TYPE (* IEC61131-3, Table 14#5 *)
  (* Standard: 1131-3 *)
  (* Version 0.0, 1/8/2024, Cheyan, Schneider Electric, Template *)
  PACKAGE Main;
  {SET_ATTRIBUTE(nxtDataType, /vixPIdCcZIb6QWPlMQZzxk/Xodw6ZTz7GLmAa8/l8jdeuo9fE+SuB4FxdXXE802R0CdcCLDo/vWly1uib6SOZYiAwivmAel2yHu1WhlYxNG8E6FaEvIshAMijy0HUFTIWQPES4Hn6O2Me7+1G8xKDYtS96nh2/xLpmfovEYUFIvpSFOGf63LdZn3qKyjU3+GSMGtmwYiPA=)}
  DPC_STATUS_CTLMODEL : STRUCT
    stVal : stVal;
    q : Quality;
    t : TimeStamp;
    CtlModel : CtlModels;
  END_STRUCT;
END_TYPE
